FUNCTION_BLOCK StopGroupTask_TestSuite
VAR
	ThisTestSuite : TestSuite<TestSuiteParameter.MaxTestCount>('C:\ProgramData\Beckhoff\TwinCAT\3.1\Boot\StopGroup_Tests.xml') := (TestSuiteName := 'StopGroup Test Suite');
END_VAR

TaskAcceptsValidCommand_Test();
TaskRejectsCommandWithNoRef_Test();
TaskRejectsCycleWithNoRef_Test();
TaskRejectsDuplicateCommand_Test();
TaskRejectsZeroDecel_Test();
TaskRejectsZeroJerk_Test();
TaskRejectsInvalidCAGroup();

METHOD TaskAcceptsValidCommand_Test
VAR
	stubCAGroup : CollisionGroup;
	testStopGrp : StopMoverGroup:= (MyCollisionGroup := stubCAGroup);
	Expected : BOOL := TRUE;
	Actual	 : BOOL;
END_VAR
IF ThisTestSuite.Test(__POUNAME()).ExecuteTest() THEN
	Actual := SUCCEEDED(testStopGrp.Execute());
	ThisTestSuite.Test(__POUNAME()).AssertEqual(Expected, Actual);
END_IF
END_METHOD

METHOD TaskRejectsCommandWithNoRef_Test
VAR
	testStopGrp : StopMoverGroup;
	Expected : BOOL := TRUE;
	Actual	 : BOOL;
END_VAR
IF ThisTestSuite.Test(__POUNAME()).ExecuteTest() THEN
	Actual := FAILED(testStopGrp.Execute());
	ThisTestSuite.Test(__POUNAME()).AssertEqual(Expected, Actual);
END_IF
END_METHOD

METHOD TaskRejectsCycleWithNoRef_Test
VAR
	testStopGrp : StopMoverGroup;
	Expected : BOOL := TRUE;
	Actual	 : BOOL;
END_VAR
IF ThisTestSuite.Test(__POUNAME()).ExecuteTest() THEN
	Actual := FAILED(testStopGrp.Cycle());
	ThisTestSuite.Test(__POUNAME()).AssertEqual(Expected, Actual);
END_IF
END_METHOD

METHOD TaskRejectsDuplicateCommand_Test
VAR
	stubCAGroup : CollisionGroup;
	testStopGrp : StopMoverGroup:= (MyCollisionGroup := stubCAGroup);
	Expected : BOOL := TRUE;
	Actual	 : BOOL;
END_VAR
IF ThisTestSuite.Test(__POUNAME()).ExecuteTest() THEN
	testStopGrp.Execute();
	Actual := FAILED(testStopGrp.Execute());
	ThisTestSuite.Test(__POUNAME()).AssertEqual(Expected, Actual);
END_IF
END_METHOD

METHOD TaskRejectsInvalidCAGroup
VAR
	stubGroup : CollisionGroup;
	iStubCAGRoup : I_CollisionGroup := stubGroup;
	testStopGrp : StopMoverGroup:= (MyCollisionGroup := stubGroup);
	Expected : BOOL := TRUE;
	Actual	 : BOOL;
END_VAR
IF ThisTestSuite.Test(__POUNAME()).ExecuteTest() THEN
	testStopGrp.MyCollisionGroup := 16#0;
	Actual := testStopGrp.MyCollisionGroup = iStubCAGroup;
	ThisTestSuite.Test(__POUNAME()).AssertEqual(Expected, Actual);
END_IF
END_METHOD

METHOD TaskRejectsZeroDecel_Test
VAR
	stubCAGroup : CollisionGroup;
	testStopGrp : StopMoverGroup:= (MyCollisionGroup := stubCAGroup);
	Expected : BOOL := TRUE;
	Actual	 : BOOL;
END_VAR
IF ThisTestSuite.Test(__POUNAME()).ExecuteTest() THEN
	testStopGrp.Deceleration := 1000.0;
	testStopGrp.Deceleration := 0.0;
	Actual := testStopGrp.Deceleration <> 0.0;
	ThisTestSuite.Test(__POUNAME()).AssertEqual(Expected, Actual);
END_IF
END_METHOD

METHOD TaskRejectsZeroJerk_Test
VAR
	stubCAGroup : CollisionGroup;
	testStopGrp : StopMoverGroup:= (MyCollisionGroup := stubCAGroup);
	Expected : BOOL := TRUE;
	Actual	 : BOOL;
END_VAR
IF ThisTestSuite.Test(__POUNAME()).ExecuteTest() THEN
	testStopGrp.Jerk := 1000.0;
	testStopGrp.Jerk := 0.0;
	Actual := testStopGrp.Jerk <> 0.0;
	ThisTestSuite.Test(__POUNAME()).AssertEqual(Expected, Actual);
END_IF
END_METHOD

END_FUNCTION_BLOCK

(* stored: Version 1.1.0.1
   POU StopGroupTask_TestSuite: Id {99aef4ad-4fc7-41c6-a957-800e5b929308}, SpecialFunc None
   Method TaskAcceptsValidCommand_Test: Id {bbbd6c90-0584-49fd-9b9a-b03e6807aed2}
   Method TaskRejectsCommandWithNoRef_Test: Id {d1ce67c8-b8c6-45a7-99fc-4bf33acd3be8}
   Method TaskRejectsCycleWithNoRef_Test: Id {ef2644e4-091e-4487-8a64-1b9096d6b7d5}
   Method TaskRejectsDuplicateCommand_Test: Id {bffcdbff-9e58-4f9c-b472-3c027ffeccec}
   Method TaskRejectsInvalidCAGroup: Id {18fb45de-e16e-44a2-89fb-912d3460aea0}
   Method TaskRejectsZeroDecel_Test: Id {2ad511e9-12d7-4d9d-9f2e-89b206f19ab8}
   Method TaskRejectsZeroJerk_Test: Id {0cdab2f7-a911-4354-b921-151032733675} *)
